// TIA Portal V19 export
TYPE "udt_LDrvSafe_typeSinaSTlg30Status"
TITLE = LDrvSafe_typeSinaSTlg30Status
// Failsafe user-defined data type for PROFIsafe telegram 30 to get status information of Safety Integrated Functions of SINAMICS S
// stored: Access Published, IsFailsafeCompliant true
   STRUCT
      STOactive { ExternalWritable := 'False'} : Bool;   // Safety Function Safe Torque Off active
      SS1active { ExternalWritable := 'False'} : Bool;   // Safety Function Safe Stop 1 active
      SS2active { ExternalWritable := 'False'} : Bool;   // Safety Function Safe Stop 2 active
      SOSactive { ExternalWritable := 'False'} : Bool;   // Safety Function Safe Operating Stop active
      SLSactive { ExternalWritable := 'False'} : Bool;   // Safety Function Safely-limited Speed active
      reserved1 { ExternalWritable := 'False'} : Bool;   // Reserve bit 1
      SLPactive { ExternalWritable := 'False'} : Bool;   // Safety Function Safely-limited Position active
      internalEvent { ExternalWritable := 'False'} : Bool;   // Internal Event occured (Safety error in SINAMICS)
      SLAactive { ExternalWritable := 'False'} : Bool;   // Safety Function Safely-limited Acceleration active
      SLSbit0Active { ExternalWritable := 'False'} : Bool;   // One of the the four SLS limits is active; operates together with bit 1
      SLSbit1Active { ExternalWritable := 'False'} : Bool;   // One of the the four SLS limits is active; operates together with bit 0
      SOSselected { ExternalWritable := 'False'} : Bool;   // Safety Function Safe Operating Stop selected (not active yet)
      SDIpositiveActive { ExternalWritable := 'False'} : Bool;   // Safety Function Safe Direction (positive direction) active
      SDInegativeActive { ExternalWritable := 'False'} : Bool;   // Safety Function Safe Direction (negative direction) active
      reserved3 { ExternalWritable := 'False'} : Bool;   // Reserve bit 3
      SSMactive { ExternalWritable := 'False'} : Bool;   // Safety Function Safe Speed Monitor; signals, if safe speed is below paramterizable speed limit
   END_STRUCT;
END_TYPE
